(* PLC project Unnamed, Unknown Unnamed 1 *)
(* stored: creationDateTime 2024-01-28T21:46:12, modificationDateTime 2024-01-28T22:24:48 *)

PROGRAM Lab1
  VAR
    PB1 AT %IX100.0 : BOOL;
    PB2 AT %IX100.1 : BOOL;
    LED AT %QX100.0 : BOOL;
  END_VAR

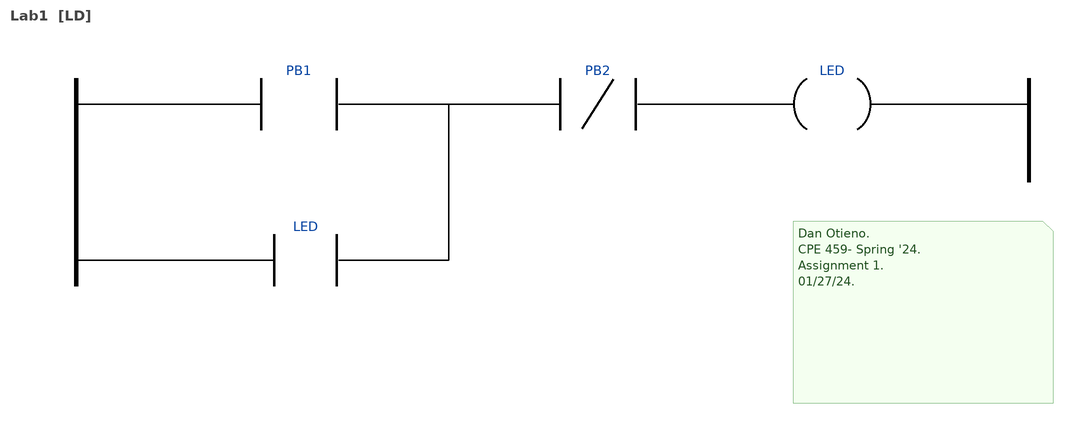
(* LD diagram, written out as Structured Text *)
LED := (PB1 OR LED) AND NOT PB2;
(* Dan Otieno.
CPE 459- Spring '24.
Assignment 1.
01/27/24. *)
END_PROGRAM

CONFIGURATION Config0
  RESOURCE Res0 ON PLC
    TASK task0(INTERVAL := T#20ms, PRIORITY := 0);
    PROGRAM instance0 WITH task0 : Lab1;
  END_RESOURCE
END_CONFIGURATION
